(* IEC 61131-3 sources: cyrus-cybernetic/, 5 files *)

(* ---- generated_plc_function_block.plc ---- *)
// Generated_FBD_Program
// Generated Function Block Diagram
// Description: Conveyor belt sequencing logic

// Function Block Network:
// Input_Start (BOOL) --> AND_Block --> Output_Motor (BOOL)
// Input_Stop (BOOL) --> AND_Block
// Emergency_Stop (BOOL) --> NOT_Block --> AND_Block

PROGRAM Generated_FBD_Program
VAR
    Input_Start AT %IX0.0 : BOOL;
    Input_Stop AT %IX0.1 : BOOL;
    Emergency_Stop AT %IX0.2 : BOOL;
    Output_Motor AT %QX0.0 : BOOL;
    AND_Block : AND;  // AND function block
    NOT_Block : NOT;  // NOT function block
END_VAR

// Connect function blocks
NOT_Block.IN := Emergency_Stop;
AND_Block.IN1 := Input_Start;
AND_Block.IN2 := NOT_Block.OUT;
Output_Motor := AND_Block.OUT;

END_PROGRAM

(* ---- generated_plc_instruction_list.plc ---- *)
// Generated_IL_Program
// Generated Instruction List Program
// Description: Basic I/O mapping and control

PROGRAM Generated_IL_Program
VAR
    Start_Button AT %IX0.0 : BOOL;
    Stop_Button AT %IX0.1 : BOOL;
    Motor_Run AT %QX0.0 : BOOL;
    Emergency_Stop AT %IX0.2 : BOOL;
END_VAR

// Instruction List Logic
LD    Start_Button      // Load Start Button
ANDN  Stop_Button       // AND NOT Stop Button
ANDN  Emergency_Stop    // AND NOT Emergency Stop
ST    Motor_Run         // Store to Motor Run

END_PROGRAM

(* ---- generated_plc_ladder.plc ---- *)
// Generated_Ladder_Program
// Generated Ladder Logic Program
// Description: Motor control with start/stop and emergency stop

PROGRAM Generated_Ladder_Program
VAR
    Start_Button AT %IX0.0 : BOOL;     // Start button input
    Stop_Button AT %IX0.1 : BOOL;      // Stop button input
    Motor_Run AT %QX0.0 : BOOL;        // Motor run output
    Emergency_Stop AT %IX0.2 : BOOL;   // Emergency stop
    Timer_Run AT %QX0.1 : BOOL;        // Timer output
    Timer_Preset : TIME := T#5S;       // 5 second timer
    Timer_Current : TIME;
END_VAR

// Ladder Rung 1: Motor Start/Stop Logic
Start_Button   Stop_Button   Emergency_Stop   Motor_Run
------| |--------| |------------| |-------------( )

// Ladder Rung 2: Timer Logic
Motor_Run      Timer_Run
------| |---------( )

// Ladder Rung 3: Timer Reset
Stop_Button    Emergency_Stop
------| |--------| |-------------( )

END_PROGRAM

(* ---- generated_plc_sequential.plc ---- *)
// Generated_SFC_Program
// Generated Sequential Function Chart
// Description: Batch process control with steps

PROGRAM Generated_SFC_Program
VAR
    Start_Command AT %IX0.0 : BOOL;
    Step_Complete AT %IX0.1 : BOOL;
    Reset_Command AT %IX0.2 : BOOL;
    Step1_Active AT %QX0.0 : BOOL;
    Step2_Active AT %QX0.1 : BOOL;
    Step3_Active AT %QX0.2 : BOOL;
END_VAR

// Sequential Function Chart
INITIAL_STEP Start:
    Step1_Active := TRUE;
END_STEP

TRANSITION Start_TO_Step1:
    Start_Command
END_TRANSITION

STEP Step1:
    // Step 1 actions
    Step1_Active := TRUE;
END_STEP

TRANSITION Step1_TO_Step2:
    Step_Complete
END_TRANSITION

STEP Step2:
    // Step 2 actions
    Step2_Active := TRUE;
END_STEP

TRANSITION Step2_TO_Step3:
    Step_Complete
END_TRANSITION

STEP Step3:
    // Step 3 actions - Final step
    Step3_Active := TRUE;
END_STEP

END_PROGRAM

(* ---- generated_plc_structured_text.plc ---- *)
// Generated_ST_Program
// Generated Structured Text Program
// Description: PID temperature control system

PROGRAM Generated_ST_Program
VAR
    Start_Button AT %IX0.0 : BOOL;
    Stop_Button AT %IX0.1 : BOOL;
    Motor_Run AT %QX0.0 : BOOL;
    Emergency_Stop AT %IX0.2 : BOOL;
    Timer_Run AT %QX0.1 : BOOL;
    Timer_Preset : TIME := T#5S;
    Timer_Current : TIME;
    Counter_Value : INT := 0;
END_VAR

// Main control logic
IF Emergency_Stop THEN
    Motor_Run := FALSE;
    Timer_Run := FALSE;
ELSIF Start_Button AND NOT Stop_Button THEN
    Motor_Run := TRUE;
    Timer_Run := TRUE;
ELSIF Stop_Button THEN
    Motor_Run := FALSE;
    Timer_Run := FALSE;
END_IF;

// Counter logic
IF Motor_Run AND Timer_Run THEN
    Counter_Value := Counter_Value + 1;
END_IF;

END_PROGRAM
